FUNCTION_BLOCK GreenMasterAIU EXTENDS GreenMasterAIU_Base
VAR_INPUT
END_VAR
VAR_OUTPUT
END_VAR
VAR
	IO_AI_09: PressureInput;
	IO_AI_10: PressureInput;
	IO_AI_11: PressureInput;
	IO_AI_12: PressureInput;
	IO_AI_13: PressureInput;
	IO_AI_14: PressureInput;
	IO_AI_15: PressureInput;
	IO_AI_16: PressureInput;
END_VAR


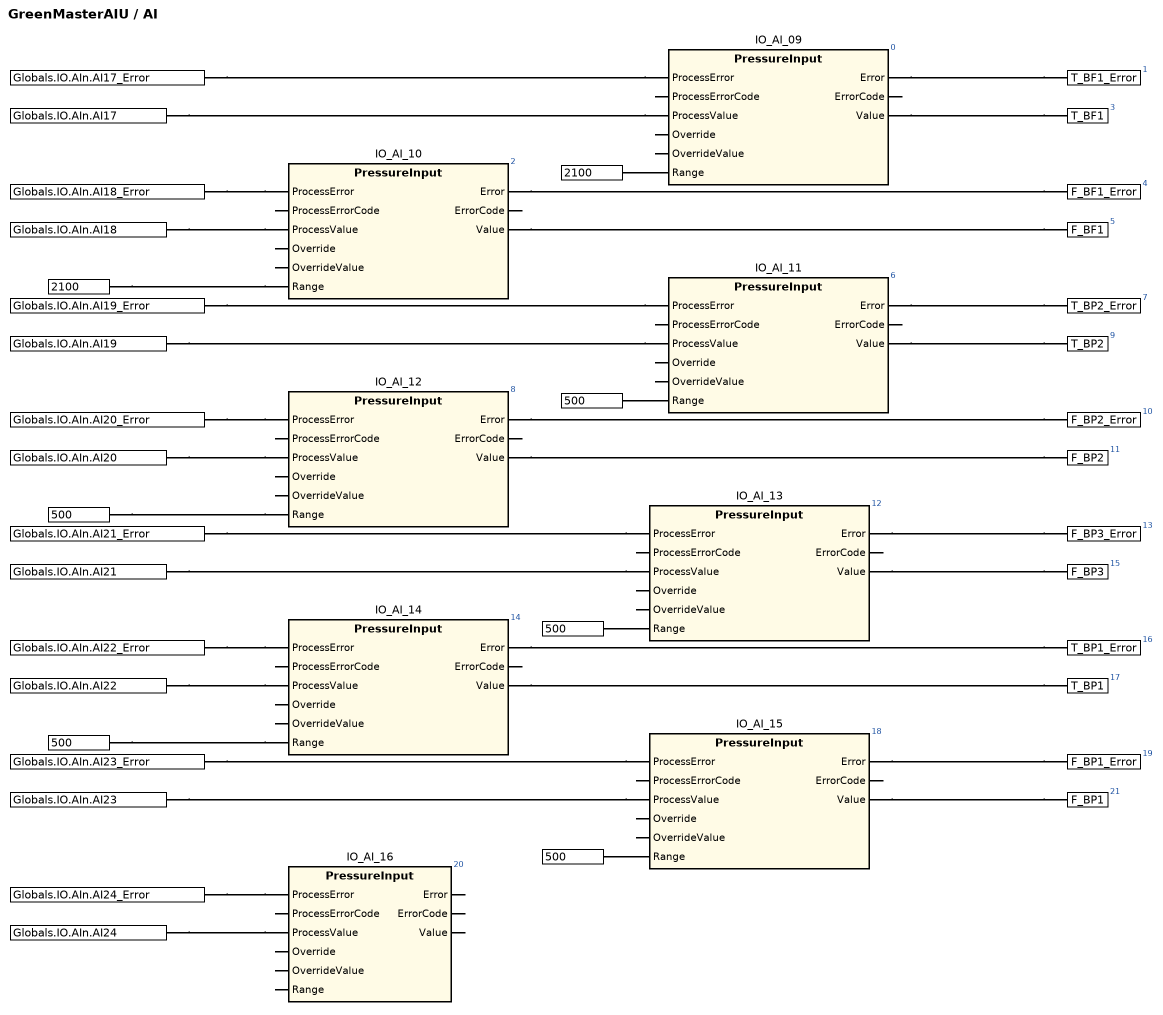
// PAGE AI
IO_AI_09(ProcessError := Globals.IO.AIn.AI17_Error, ProcessValue := Globals.IO.AIn.AI17, Range := 2100); // PressureInput
T_BF1_Error := IO_AI_09.Error;
IO_AI_10(ProcessError := Globals.IO.AIn.AI18_Error, ProcessValue := Globals.IO.AIn.AI18, Range := 2100); // PressureInput
T_BF1 := IO_AI_09.Value;
F_BF1_Error := IO_AI_10.Error;
F_BF1 := IO_AI_10.Value;
IO_AI_11(ProcessError := Globals.IO.AIn.AI19_Error, ProcessValue := Globals.IO.AIn.AI19, Range := 500); // PressureInput
T_BP2_Error := IO_AI_11.Error;
IO_AI_12(ProcessError := Globals.IO.AIn.AI20_Error, ProcessValue := Globals.IO.AIn.AI20, Range := 500); // PressureInput
T_BP2 := IO_AI_11.Value;
F_BP2_Error := IO_AI_12.Error;
F_BP2 := IO_AI_12.Value;
IO_AI_13(ProcessError := Globals.IO.AIn.AI21_Error, ProcessValue := Globals.IO.AIn.AI21, Range := 500); // PressureInput
F_BP3_Error := IO_AI_13.Error;
IO_AI_14(ProcessError := Globals.IO.AIn.AI22_Error, ProcessValue := Globals.IO.AIn.AI22, Range := 500); // PressureInput
F_BP3 := IO_AI_13.Value;
T_BP1_Error := IO_AI_14.Error;
T_BP1 := IO_AI_14.Value;
IO_AI_15(ProcessError := Globals.IO.AIn.AI23_Error, ProcessValue := Globals.IO.AIn.AI23, Range := 500); // PressureInput
F_BP1_Error := IO_AI_15.Error;
IO_AI_16(ProcessError := Globals.IO.AIn.AI24_Error, ProcessValue := Globals.IO.AIn.AI24); // PressureInput
F_BP1 := IO_AI_15.Value;

END_FUNCTION_BLOCK

(* stored: Version 1.1.0.1, ProductVersion 3.1.4024.6
   POU GreenMasterAIU: Id {e17068a2-f508-4c64-b743-5a3e494a702d}, SpecialFunc None *)
